# EPICS autosave request: auto_settings.req
$(Sys)$(Dev)V-R
$(Sys)$(Dev)V-SF
